FUNCTION_BLOCK ClampInsertion EXTENDS Insertion
VAR
	slider : ServoNC;
	screw : TeknicEIP;
END_VAR

slider(
	bEnable:= enable, 
	home=> , 
	outerLimit=> , 
	innerLimit=> , 
	ready=> , 
	busy=> , 
	error=> , 
	homeSet=> , 
	position=> sliderPos);

screw(
	bEnable:= enable, 
	home=> , 
	outerLimit=> , 
	innerLimit=> , 
	done=> , 
	homeSet=> , 
	busy=> , 
	error=> , 
	position=> screwPos);

home := screw.home AND slider.home;
busy := slider.busy OR screw.busy;
error := slider.error OR screw.error;

METHOD align : BOOL
VAR_INPUT
	targetPos : REAL;
END_VAR
align := slider.moveAbsolute(targetPos := targetPos);
END_METHOD

METHOD homingSequence : BOOL
IF NOT slider.homeSet THEN
	slider.homingSequence();
END_IF

IF NOT screw.homeSet THEN
	screw.homingSequence();
END_IF

homingSequence := slider.homeSet AND screw.homeSet;
END_METHOD

METHOD press : BOOL
screw.moveContinuous(direction := MC_Negative_Direction);
END_METHOD

METHOD release : BOOL
VAR_INPUT
END_VAR
screw.moveContinuous(direction := MC_Positive_Direction);
END_METHOD

METHOD traverse : BOOL
VAR_INPUT
	direction : MC_Direction;
END_VAR
slider.moveContinuous(direction := direction);
END_METHOD

END_FUNCTION_BLOCK

(* stored: Version 1.1.0.1, ProductVersion 3.1.4024.11
   POU ClampInsertion: Id {5863597f-27b0-4dbc-9d04-6ecef8e924c0}, SpecialFunc None
   Method align: Id {cb86c80e-0707-465a-8508-1718a96c3419}
   Method homingSequence: Id {e67f0be0-54d4-462b-b379-345eff57e103}
   Method press: Id {56522197-b622-4b8a-97a4-2f6f5b1e037d}
   Method release: Id {32d29e49-2530-44bf-b36b-1459e8c3dd33}
   Method traverse: Id {c602204b-17a2-4d87-a4b6-22c50ab42546} *)
